PROGRAM MAIN
VAR
	TestTester		: TestTester;
	ReRun			: BOOL;
	ReRunSingleTest : BOOL;
END_VAR

TestSuite.TestSuiteName := 'My Test Test-Suite';
Test_Counter_AddTwo();
Test_Counter_SubtractTwo();
Test_Bool();
Test_String();
Test_Lreal();
Test_Real();
SecondTestSuite();
TestSuiteOverflow();
IF ReRun THEN
	TestSuite.ReRunTests();
	ReRun := FALSE;
END_IF

IF ReRunSingleTest THEN
	TestSuite.ReRunIndividualTest('MAIN.Test_Counter_AddTwo');
	ReRunSingleTest := FALSE;
END_IF

METHOD Test_Bool
VAR_INST
	Expected : BOOL;
	Actual	 : BOOL;
END_VAR
IF TestSuite.Test(__POUNAME()).ExecuteTest() THEN
	Expected := TRUE;
	Actual	 := TestTester.TestBool;
	TestSuite.Test(__POUNAME()).AssertEqual(Expected, Actual);
END_IF
END_METHOD

METHOD Test_Counter_AddTwo
VAR_INST
	Expected : DINT;
	Actual	 : DINT;
END_VAR
IF TestSuite.Test(__POUNAME()).ExecuteTest() THEN
	Expected := 10;
	Actual	 := TestTester.AddTwo(5, 5);
	TestSuite.Test(__POUNAME()).AssertEqual(Expected, Actual);
END_IF
END_METHOD

METHOD Test_Counter_SubtractTwo
VAR_INST
	Expected : DINT;
	Actual	 : DINT;
END_VAR
IF TestSuite.Test(__POUNAME()).ExecuteTest() THEN
	Expected := 0;
	Actual	 := TestTester.AddTwo(5, -5);
	TestSuite.Test(__POUNAME()).AssertEqual(Expected, Actual);
END_IF
END_METHOD

METHOD Test_Lreal
VAR_INST
	Expected : LREAL;
	Actual	 : LREAL;
END_VAR
IF TestSuite.Test(__POUNAME()).ExecuteTest() THEN
	Expected := 75.75;
	Actual	 := TestTester.TestLReal;
	TestSuite.Test(__POUNAME()).AssertEqual(Expected, Actual, 0.1);
END_IF
END_METHOD

METHOD Test_Real
VAR_INST
	Expected : REAL;
	Actual	 : REAL;
END_VAR
IF TestSuite.Test(__POUNAME()).ExecuteTest() THEN
	Expected := 75.75;
	Actual	 := TestTester.TestLReal;
	TestSuite.Test(__POUNAME()).AssertEqual(Expected, Actual, 0.1);
END_IF
END_METHOD

METHOD Test_String
VAR_INST
	Expected : STRING;
	Actual	 : STRING;
END_VAR
VAR
    SizeString : DINT;
END_VAR
IF TestSuite.Test(__POUNAME()).ExecuteTest() THEN
	Expected := 'TestString';
	Actual	 := TestTester.TestString;
	TestSuite.Test(__POUNAME()).AssertEqual(Expected, Actual);
END_IF
END_METHOD

END_PROGRAM

(* stored: Version 1.1.0.1
   POU MAIN: Id {7dbbc5fe-66aa-4f70-a8be-dd1553a601dc}, SpecialFunc None
   Method Test_Bool: Id {0a23e9d2-f7ab-4c19-9735-98437bc044ae}
   Method Test_Counter_AddTwo: Id {3d2e2d40-a28e-4d42-ab9e-06275a7cf9a4}
   Method Test_Counter_SubtractTwo: Id {82b2956c-4118-427f-a450-a3e1dcc4c03a}
   Method Test_Lreal: Id {266c5293-e490-4751-a35d-7ca22f784c01}
   Method Test_Real: Id {bbcc2c62-b42d-486a-8ed5-5d1304721b84}
   Method Test_String: Id {8bbef3dd-ba77-496f-9525-8caeed7f5a8b} *)
